Staubli VAL3: kill.pgx

public program kill()
  local string l_sMessage
begin
  call kernel:_kill()
end
